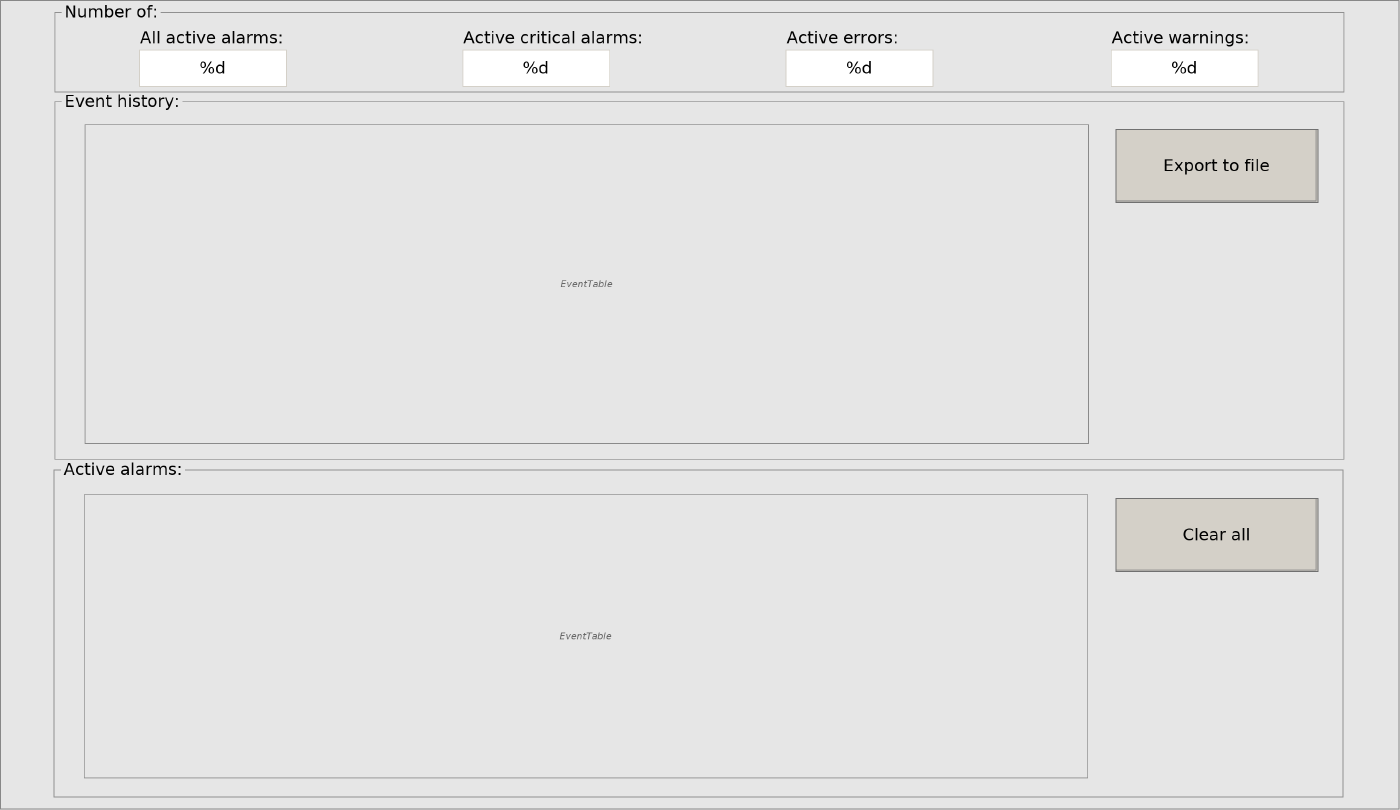
VISUALIZATION PageAlarms_1  // 1520x880
VAR_IN_OUT
	btnClearAllAlarms 	: BOOL;
	btnExportEvents		: BOOL;
	iActiveAlarms		: UDINT;
	iActiveCritical		: UDINT;
	iActiveErrors		: UDINT;
	iActiveWarrnings	: UDINT;
	arrEvents			: ARRAY[1..PSE_UniversalBlocks.iMAX_EVENTS] OF ST_Event;
	arrAlarms			: ARRAY[1..PSE_UniversalBlocks.iMAX_EVENTS] OF ST_Event;
END_VAR
    GroupBox (58,502 1400x364), "Active alarms:"
        Frame (33,35 1090x308)
            shows EventTable(data := arrAlarms)
        Button (1153,39 220x80), "Clear all"
            tap btnClearAllAlarms
    GroupBox (59,5 1400x95), "Number of:"
        Label (90,21 210x30), "All active alarms:"
        Textfield (92,49 160x40), "%d", text variable: iActiveAlarms, text list: ''
        Label (441,21 234x30), "Active critical alarms:"
        Textfield (443,49 160x40), "%d", text variable: iActiveCritical, text list: ''
        Label (792,21 210x30), "Active errors:"
        Label (1145,21 210x30), "Active warnings:"
        Textfield (794,49 160x40), "%d", text variable: iActiveErrors, text list: ''
        Textfield (1147,49 160x40), "%d", text variable: iActiveWarrnings, text list: ''
    GroupBox (59,102 1400x397), "Event history:"
        Frame (33,33 1090x347)
            shows EventTable(data := arrEvents)
        Button (1152,38 220x80), "Export to file"
            tap btnExportEvents
END_VISUALIZATION

(* stored: Version 1.1.0.1, ProductVersion 3.1.4024.12
   Visu PageAlarms_1: Id {99f0929a-0154-431f-853d-254099b6103d} *)
